(* Logix 5000 project; controller STAT 1756-L72 rev 20.12; software revision 20.04; part 16 of 34 *)
(* tags used below, declared in another part *)
   averflowput1 : DINT;
   averflowput2 : DINT;
   averK1 : DINT;
   averK2 : DINT;
   averL1 : DINT;
   averL2 : DINT;
   averL3 : DINT;
   averlpmpput2 : DINT;
   averpmpput1 : DINT;
   averQ1 : DINT;
   averQ2 : DINT;
   B16 : DINT[30];
   B17 : DINT[30];
   B3 : DINT[256];
   B9 : DINT[40];
   DateTime : DINT[7];   // DINT array tag for retrieve wallclock time through GSV created during conversion
   F8 : REAL[256];
   I19_000_Bit12 : ALIAS FOR I19[0].12;   // pulse puit put 1
   I19_000_Bit13 : ALIAS FOR I19[0].13;   // puit put 2
   I8_000_Bit09 : ALIAS FOR I8[0].9;   // midden niveau kuip 1 voorb. polyelectrolute
   I8_000_Bit10 : ALIAS FOR I8[0].10;   // hoog niveau kuip 1 voorb. polyelectrolute
   I8_000_Bit12 : ALIAS FOR I8[0].12;   // midden niveau kuip 2 voorb. polyelectrolute
   I8_000_Bit13 : ALIAS FOR I8[0].13;   // hoog niveau pekel
   N12 : DINT[230];
   N13 : DINT[230];
   N26 : DINT[256];
   O18_001_Bit02 : ALIAS FOR O18[1].2;   // pmp put 2
   O18_001_Bit04 : ALIAS FOR O18[1].4;   // PMP PUT 1
   pmpput1 : BOOL;
   pmpput2 : BOOL;
   T4 : TIMER[200];
   tot_put_1 : DINT;
   tot_put_2 : DINT;
(* ibt, continued *)

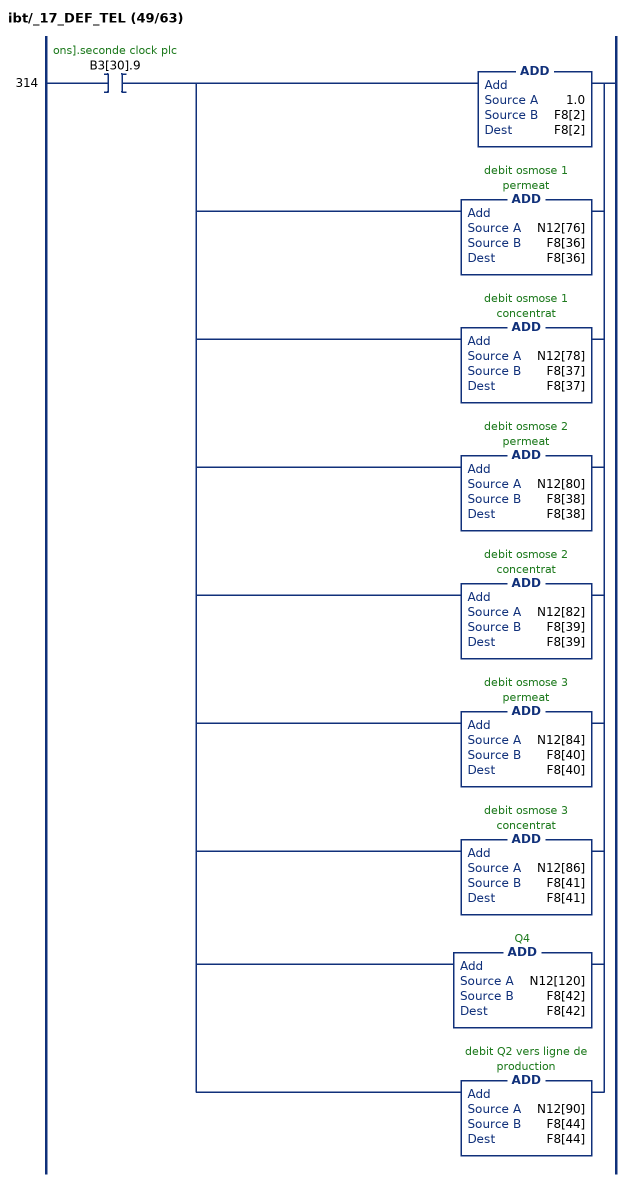
   [picture p273: ibt/_17_DEF_TEL rungs 314-314]
   314: XIC(B3[30].9)[ADD(1.0,F8[2],F8[2]) ,ADD(N12[76],F8[36],F8[36]) ,ADD(N12[78],F8[37],F8[37]) ,ADD(N12[80],F8[38],F8[38]) ,ADD(N12[82],F8[39],F8[39]) ,ADD(N12[84],F8[40],F8[40]) ,ADD(N12[86],F8[41],F8[41]) ,ADD(N12[120],F8[42],F8[42]) ,ADD(N12[90],F8[44],F8[44]) ];
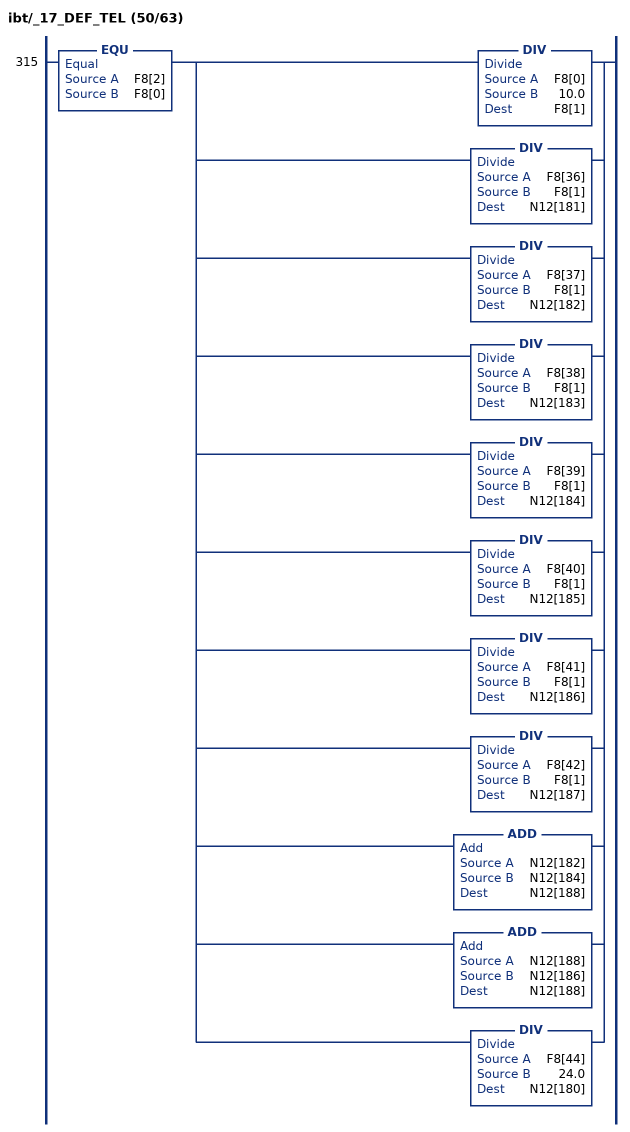
   315: EQU(F8[2],F8[0])[DIV(F8[0],10.0,F8[1]) ,DIV(F8[36],F8[1],N12[181]) ,DIV(F8[37],F8[1],N12[182]) ,DIV(F8[38],F8[1],N12[183]) ,DIV(F8[39],F8[1],N12[184]) ,DIV(F8[40],F8[1],N12[185]) ,DIV(F8[41],F8[1],N12[186]) ,DIV(F8[42],F8[1],N12[187]) ,ADD(N12[182],N12[184],N12[188]) ,ADD(N12[188],N12[186],N12[188]) ,DIV(F8[44],24.0,N12[180]) ];
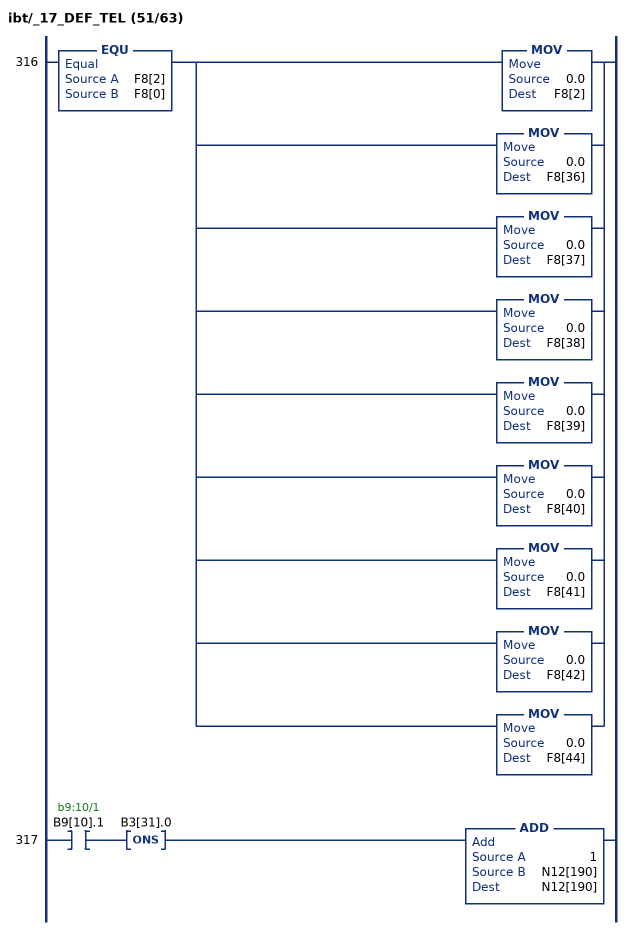
   316: EQU(F8[2],F8[0])[MOV(0.0,F8[2]) ,MOV(0.0,F8[36]) ,MOV(0.0,F8[37]) ,MOV(0.0,F8[38]) ,MOV(0.0,F8[39]) ,MOV(0.0,F8[40]) ,MOV(0.0,F8[41]) ,MOV(0.0,F8[42]) ,MOV(0.0,F8[44]) ];
   317: XIC(B9[10].1)ONS(B3[31].0)ADD(1,N12[190],N12[190]);
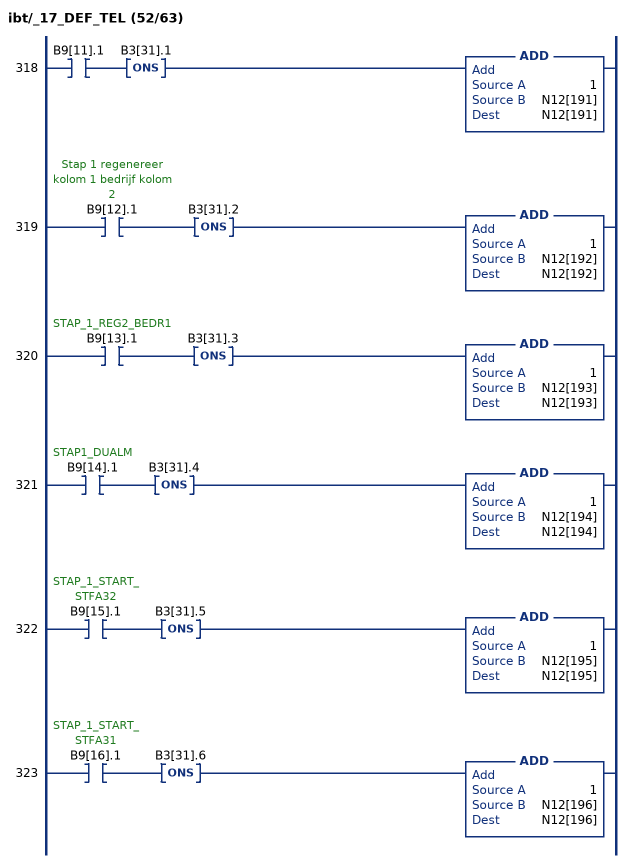
   318: XIC(B9[11].1)ONS(B3[31].1)ADD(1,N12[191],N12[191]);
   319: XIC(B9[12].1)ONS(B3[31].2)ADD(1,N12[192],N12[192]);
   320: XIC(B9[13].1)ONS(B3[31].3)ADD(1,N12[193],N12[193]);
   321: XIC(B9[14].1)ONS(B3[31].4)ADD(1,N12[194],N12[194]);
   322: XIC(B9[15].1)ONS(B3[31].5)ADD(1,N12[195],N12[195]);
   323: XIC(B9[16].1)ONS(B3[31].6)ADD(1,N12[196],N12[196]);
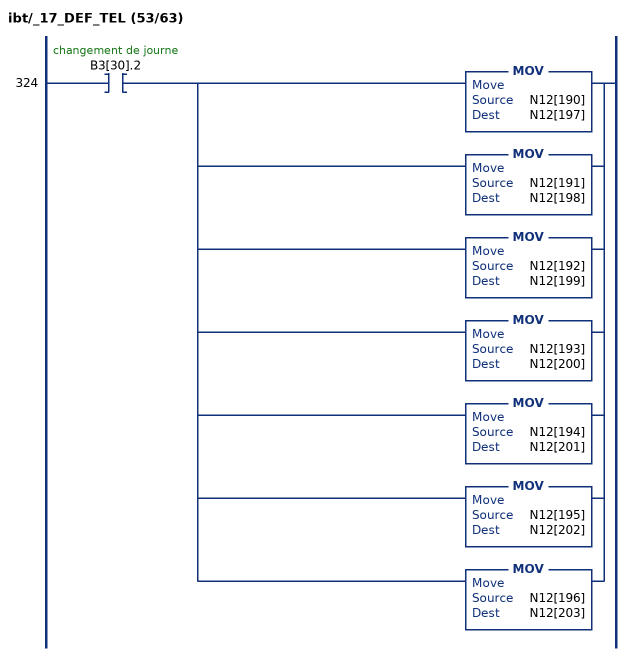
   324: XIC(B3[30].2)[MOV(N12[190],N12[197]) ,MOV(N12[191],N12[198]) ,MOV(N12[192],N12[199]) ,MOV(N12[193],N12[200]) ,MOV(N12[194],N12[201]) ,MOV(N12[195],N12[202]) ,MOV(N12[196],N12[203]) ];
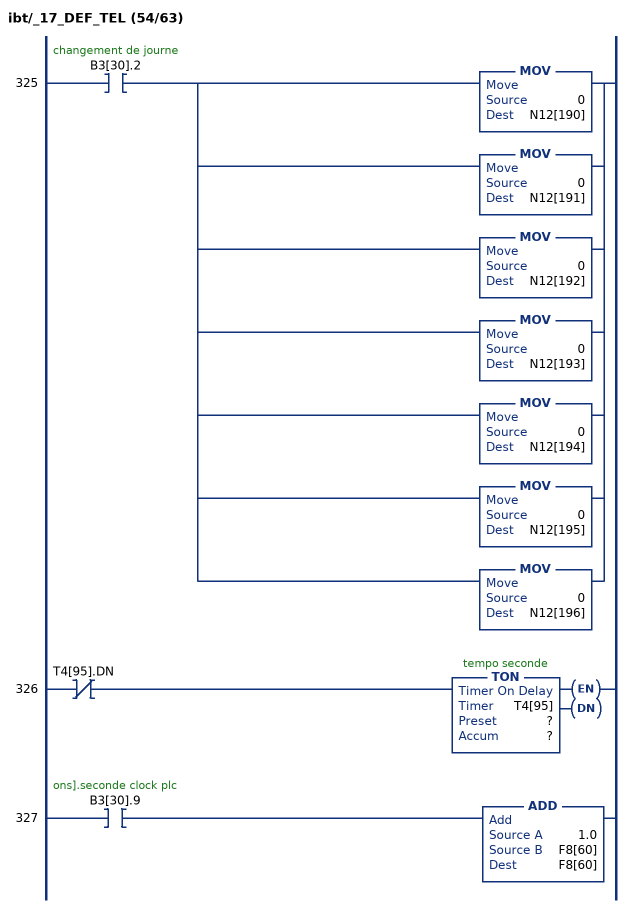
   325: XIC(B3[30].2)[MOV(0,N12[190]) ,MOV(0,N12[191]) ,MOV(0,N12[192]) ,MOV(0,N12[193]) ,MOV(0,N12[194]) ,MOV(0,N12[195]) ,MOV(0,N12[196]) ];
   326: XIO(T4[95].DN)TON(T4[95],?,?);
   327: XIC(B3[30].9)ADD(1.0,F8[60],F8[60]);
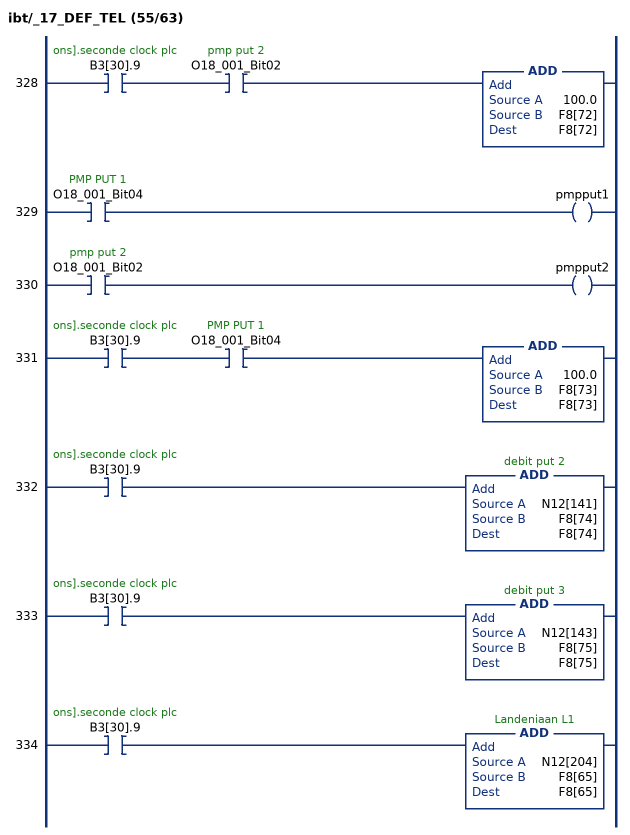
   328: XIC(B3[30].9)XIC(O18_001_Bit02)ADD(100.0,F8[72],F8[72]);
   329: XIC(O18_001_Bit04)OTE(pmpput1);
   330: XIC(O18_001_Bit02)OTE(pmpput2);
   331: XIC(B3[30].9)XIC(O18_001_Bit04)ADD(100.0,F8[73],F8[73]);
   332: XIC(B3[30].9)ADD(N12[141],F8[74],F8[74]);
   333: XIC(B3[30].9)ADD(N12[143],F8[75],F8[75]);
   334: XIC(B3[30].9)ADD(N12[204],F8[65],F8[65]);
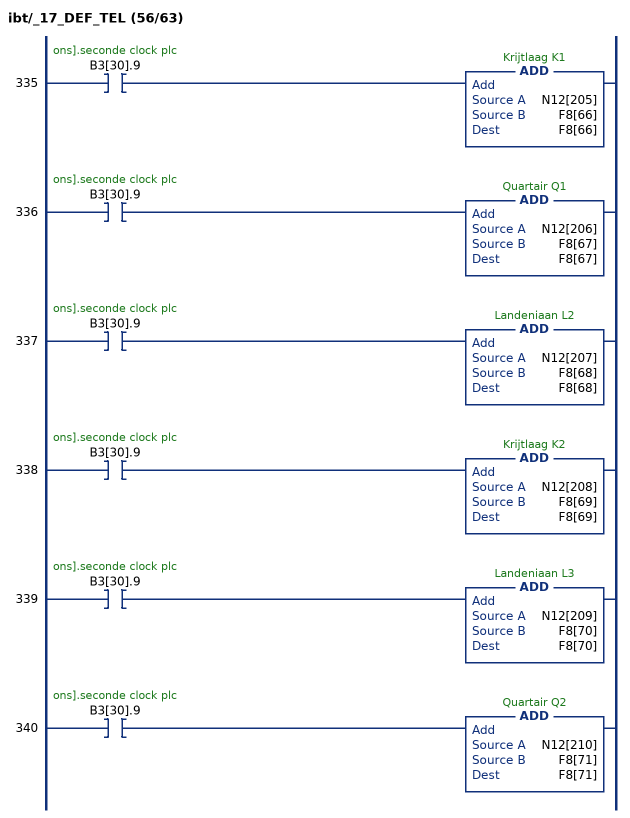
   335: XIC(B3[30].9)ADD(N12[205],F8[66],F8[66]);
   336: XIC(B3[30].9)ADD(N12[206],F8[67],F8[67]);
   337: XIC(B3[30].9)ADD(N12[207],F8[68],F8[68]);
   338: XIC(B3[30].9)ADD(N12[208],F8[69],F8[69]);
   339: XIC(B3[30].9)ADD(N12[209],F8[70],F8[70]);
   340: XIC(B3[30].9)ADD(N12[210],F8[71],F8[71]);
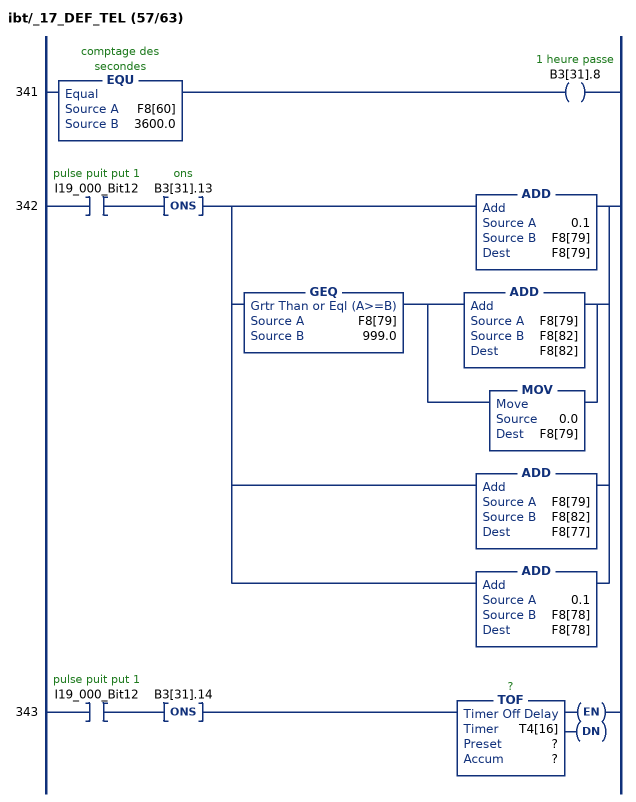
   341: EQU(F8[60],3600.0)OTE(B3[31].8);
   342: XIC(I19_000_Bit12)ONS(B3[31].13)[ADD(0.1,F8[79],F8[79]) ,GEQ(F8[79],999.0) [ADD(F8[79],F8[82],F8[82]) ,MOV(0.0,F8[79]) ] ,ADD(F8[79],F8[82],F8[77]) ,ADD(0.1,F8[78],F8[78]) ];
   343: XIC(I19_000_Bit12)ONS(B3[31].14)TOF(T4[16],?,?);
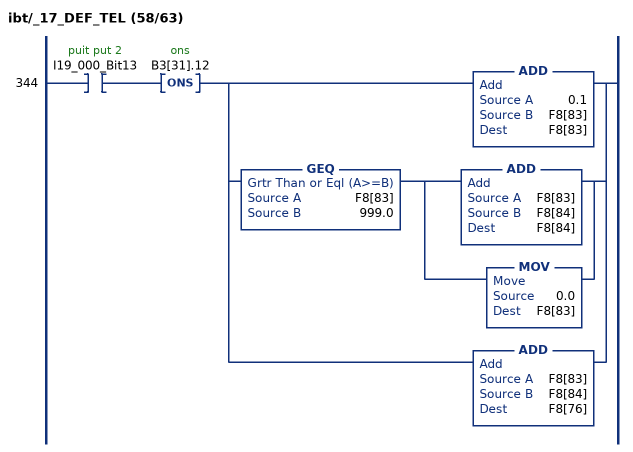
   344: XIC(I19_000_Bit13)ONS(B3[31].12)[ADD(0.1,F8[83],F8[83]) ,GEQ(F8[83],999.0) [ADD(F8[83],F8[84],F8[84]) ,MOV(0.0,F8[83]) ] ,ADD(F8[83],F8[84],F8[76]) ];
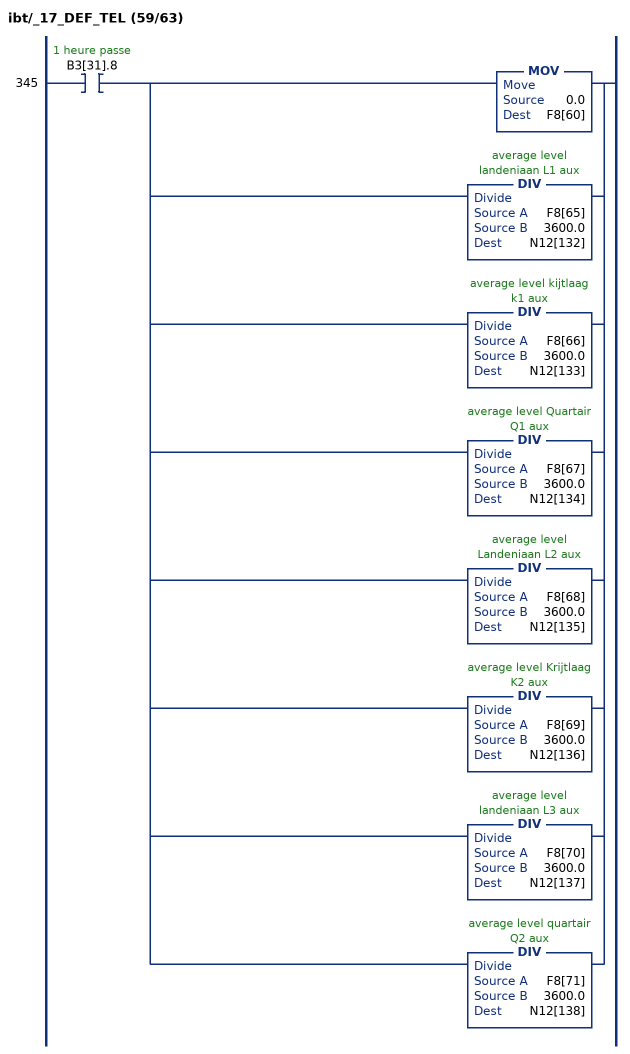
   345: XIC(B3[31].8)[MOV(0.0,F8[60]) ,DIV(F8[65],3600.0,N12[132]) ,DIV(F8[66],3600.0,N12[133]) ,DIV(F8[67],3600.0,N12[134]) ,DIV(F8[68],3600.0,N12[135]) ,DIV(F8[69],3600.0,N12[136]) ,DIV(F8[70],3600.0,N12[137]) ,DIV(F8[71],3600.0,N12[138]) ];
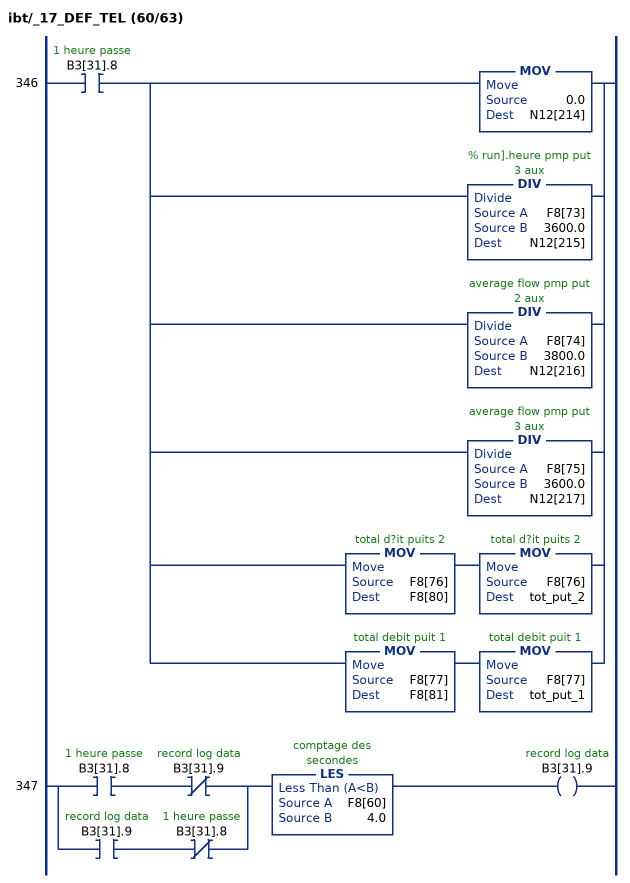
   346: XIC(B3[31].8)[MOV(0.0,N12[214]) ,DIV(F8[73],3600.0,N12[215]) ,DIV(F8[74],3800.0,N12[216]) ,DIV(F8[75],3600.0,N12[217]) ,MOV(F8[76],F8[80]) MOV(F8[76],tot_put_2) ,MOV(F8[77],F8[81]) MOV(F8[77],tot_put_1) ];
   347: [XIC(B3[31].8) XIO(B3[31].9) ,XIC(B3[31].9) XIO(B3[31].8) ]LES(F8[60],4.0)OTE(B3[31].9);
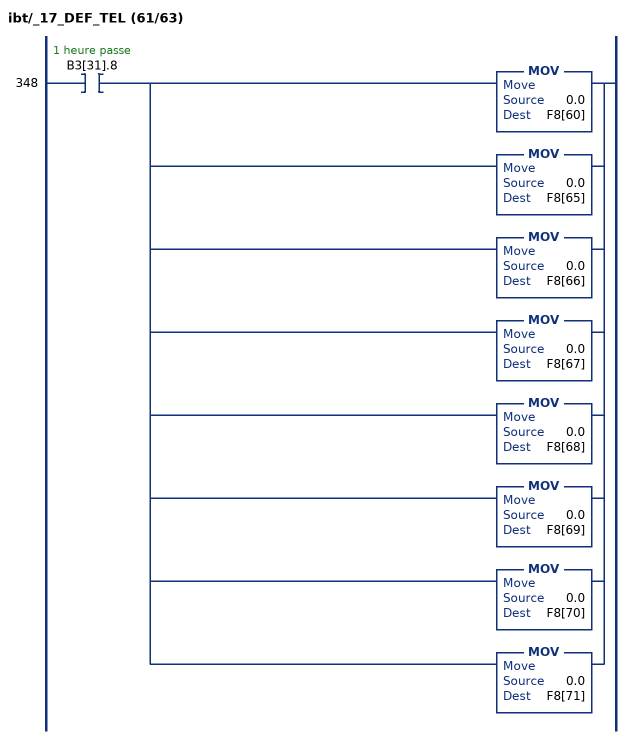
   348: XIC(B3[31].8)[MOV(0.0,F8[60]) ,MOV(0.0,F8[65]) ,MOV(0.0,F8[66]) ,MOV(0.0,F8[67]) ,MOV(0.0,F8[68]) ,MOV(0.0,F8[69]) ,MOV(0.0,F8[70]) ,MOV(0.0,F8[71]) ];
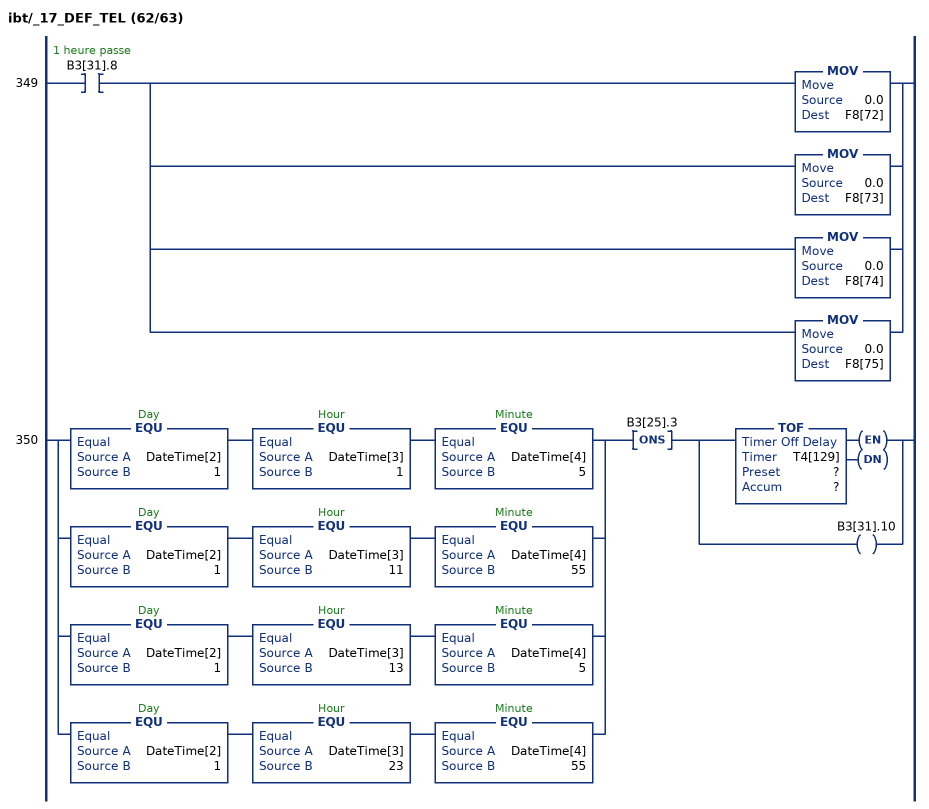
   349: XIC(B3[31].8)[MOV(0.0,F8[72]) ,MOV(0.0,F8[73]) ,MOV(0.0,F8[74]) ,MOV(0.0,F8[75]) ];
   350: [EQU(DateTime[2],1) EQU(DateTime[3],1) EQU(DateTime[4],5) ,EQU(DateTime[2],1) EQU(DateTime[3],11) EQU(DateTime[4],55) ,EQU(DateTime[2],1) EQU(DateTime[3],13) EQU(DateTime[4],5) ,EQU(DateTime[2],1) EQU(DateTime[3],23) EQU(DateTime[4],55) ]ONS(B3[25].3)[TOF(T4[129],?,?) ,OTE(B3[31].10) ];
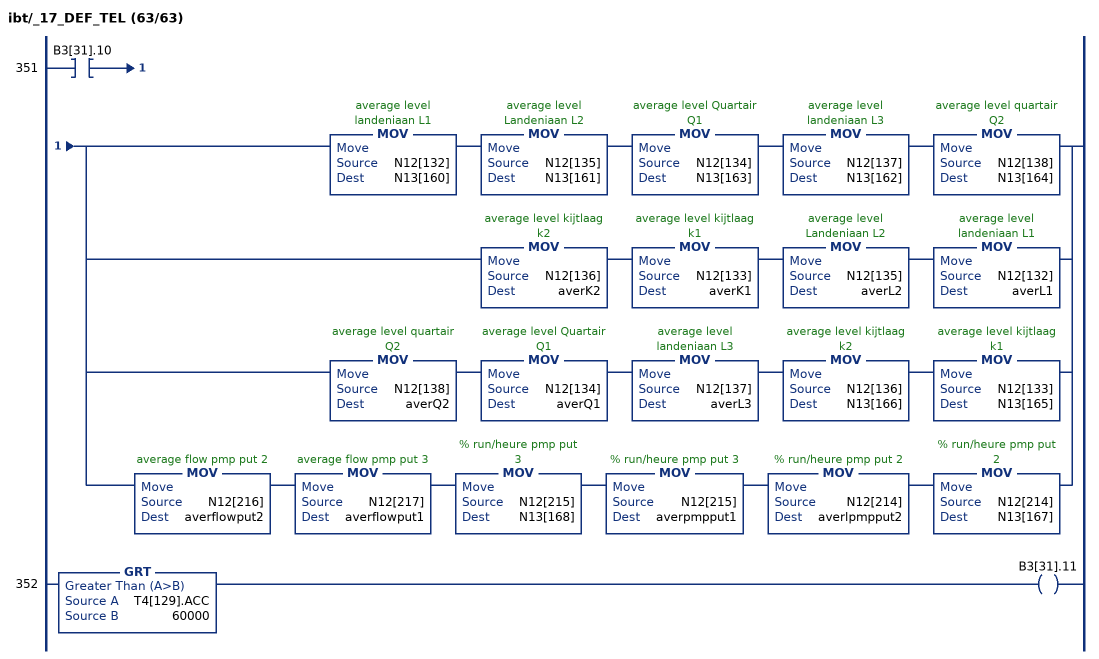
   351: XIC(B3[31].10)[MOV(N12[132],N13[160]) MOV(N12[135],N13[161]) MOV(N12[134],N13[163]) MOV(N12[137],N13[162]) MOV(N12[138],N13[164]) ,MOV(N12[136],averK2) MOV(N12[133],averK1) MOV(N12[135],averL2) MOV(N12[132],averL1) ,MOV(N12[138],averQ2) MOV(N12[134],averQ1) MOV(N12[137],averL3) MOV(N12[136],N13[166]) MOV(N12[133],N13[165]) ,MOV(N12[216],averflowput2) MOV(N12[217],averflowput1) MOV(N12[215],N13[168]) MOV(N12[215],averpmpput1) MOV(N12[214],averlpmpput2) MOV(N12[214],N13[167]) ];
   352: GRT(T4[129].ACC,60000)OTE(B3[31].11);
END_ROUTINE

ROUTINE _18_PAS_REI_Z   (* ladder *)
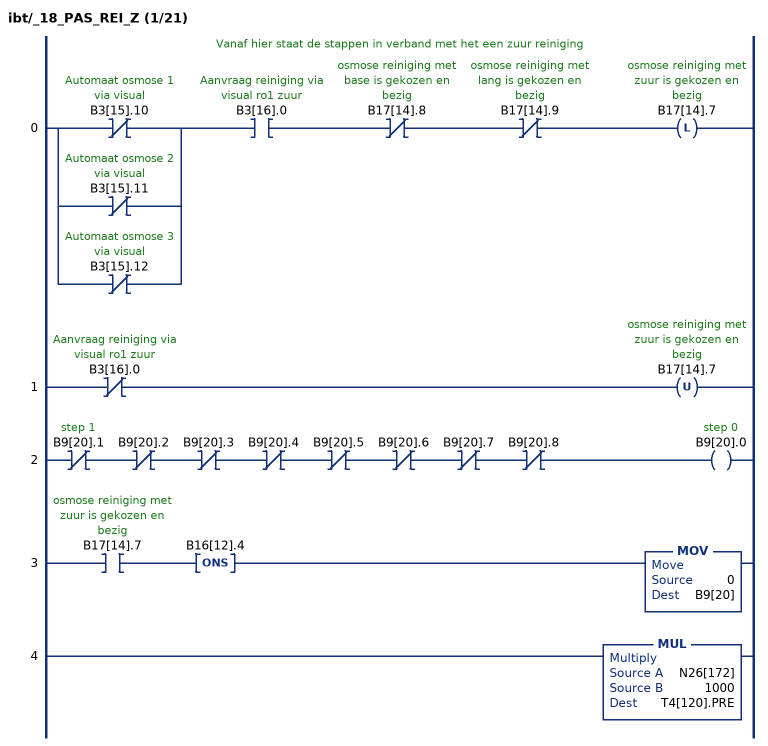
   // Vanaf hier staat de stappen in verband met het een zuur reiniging
   0: [XIO(B3[15].10) ,[XIO(B3[15].11) ,XIO(B3[15].12) ] ]XIC(B3[16].0)XIO(B17[14].8)XIO(B17[14].9)OTL(B17[14].7);
   1: XIO(B3[16].0)OTU(B17[14].7);
   2: XIO(B9[20].1)XIO(B9[20].2)XIO(B9[20].3)XIO(B9[20].4)XIO(B9[20].5)XIO(B9[20].6)XIO(B9[20].7)XIO(B9[20].8)OTE(B9[20].0);
   3: XIC(B17[14].7)ONS(B16[12].4)MOV(0,B9[20]);
   4: MUL(N26[172],1000,T4[120].PRE);
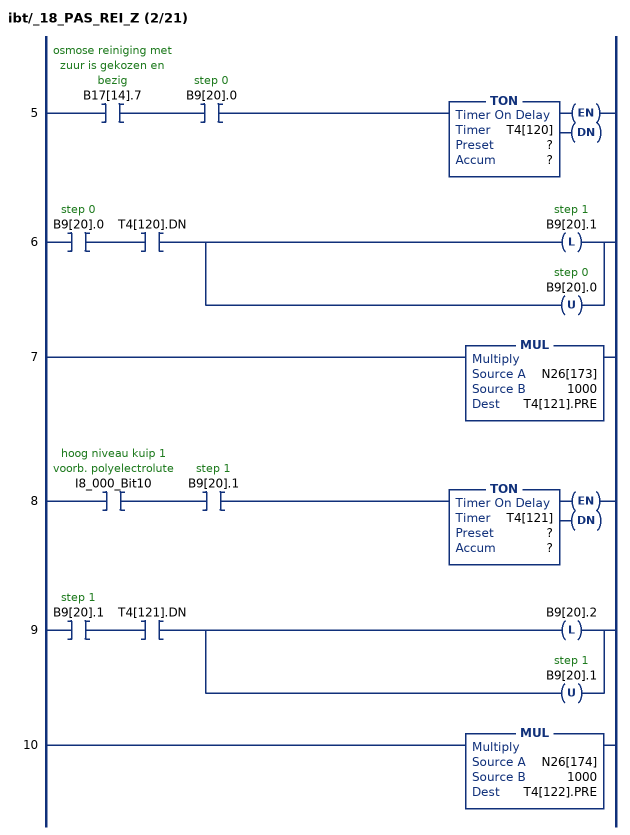
   5: XIC(B17[14].7)XIC(B9[20].0)TON(T4[120],?,?);
   6: XIC(B9[20].0)XIC(T4[120].DN)[OTL(B9[20].1) ,OTU(B9[20].0) ];
   7: MUL(N26[173],1000,T4[121].PRE);
   8: XIC(I8_000_Bit10)XIC(B9[20].1)TON(T4[121],?,?);
   9: XIC(B9[20].1)XIC(T4[121].DN)[OTL(B9[20].2) ,OTU(B9[20].1) ];
   10: MUL(N26[174],1000,T4[122].PRE);
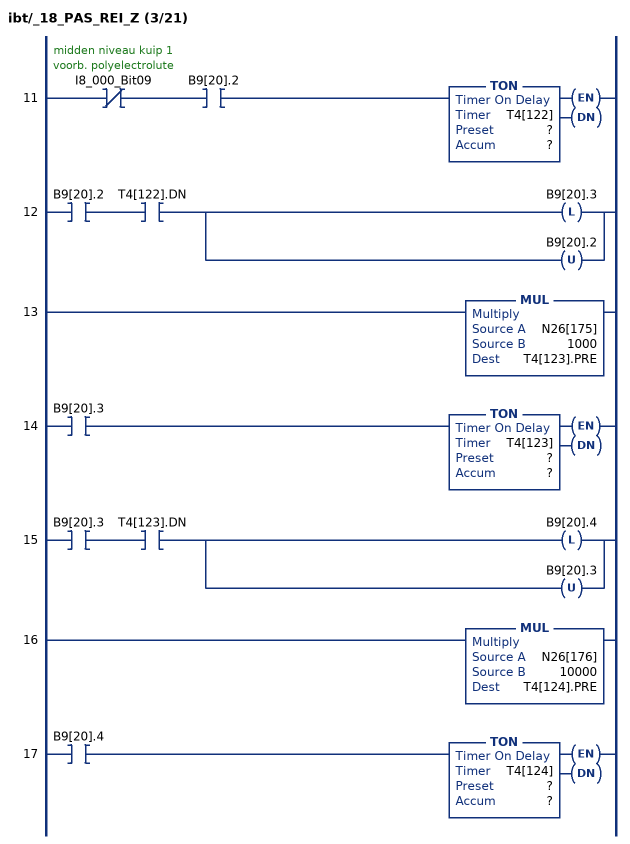
   11: XIO(I8_000_Bit09)XIC(B9[20].2)TON(T4[122],?,?);
   12: XIC(B9[20].2)XIC(T4[122].DN)[OTL(B9[20].3) ,OTU(B9[20].2) ];
   13: MUL(N26[175],1000,T4[123].PRE);
   14: XIC(B9[20].3)TON(T4[123],?,?);
   15: XIC(B9[20].3)XIC(T4[123].DN)[OTL(B9[20].4) ,OTU(B9[20].3) ];
   16: MUL(N26[176],10000,T4[124].PRE);
   17: XIC(B9[20].4)TON(T4[124],?,?);
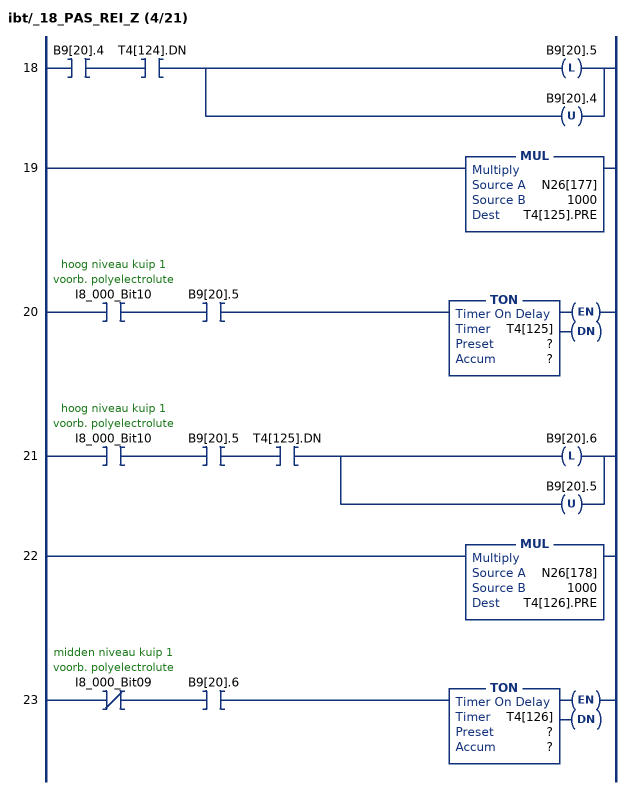
   18: XIC(B9[20].4)XIC(T4[124].DN)[OTL(B9[20].5) ,OTU(B9[20].4) ];
   19: MUL(N26[177],1000,T4[125].PRE);
   20: XIC(I8_000_Bit10)XIC(B9[20].5)TON(T4[125],?,?);
   21: XIC(I8_000_Bit10)XIC(B9[20].5)XIC(T4[125].DN)[OTL(B9[20].6) ,OTU(B9[20].5) ];
   22: MUL(N26[178],1000,T4[126].PRE);
   23: XIO(I8_000_Bit09)XIC(B9[20].6)TON(T4[126],?,?);
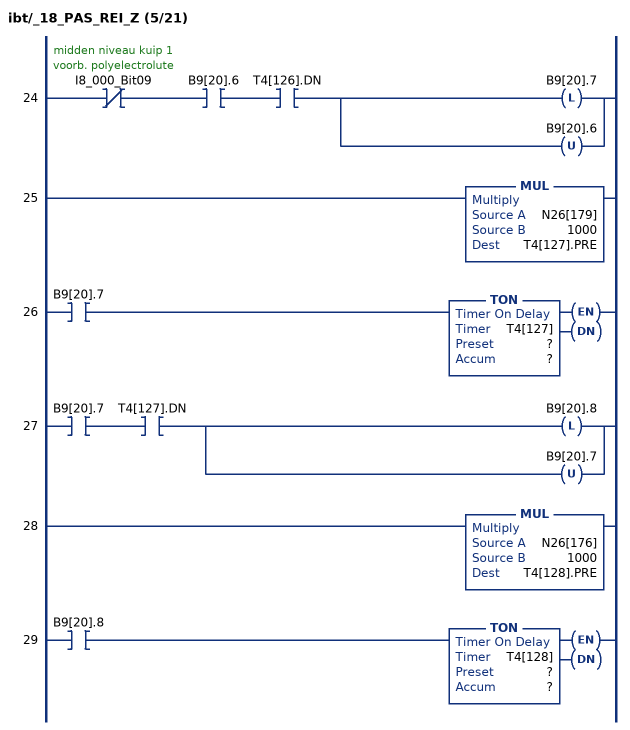
   24: XIO(I8_000_Bit09)XIC(B9[20].6)XIC(T4[126].DN)[OTL(B9[20].7) ,OTU(B9[20].6) ];
   25: MUL(N26[179],1000,T4[127].PRE);
   26: XIC(B9[20].7)TON(T4[127],?,?);
   27: XIC(B9[20].7)XIC(T4[127].DN)[OTL(B9[20].8) ,OTU(B9[20].7) ];
   28: MUL(N26[176],1000,T4[128].PRE);
   29: XIC(B9[20].8)TON(T4[128],?,?);
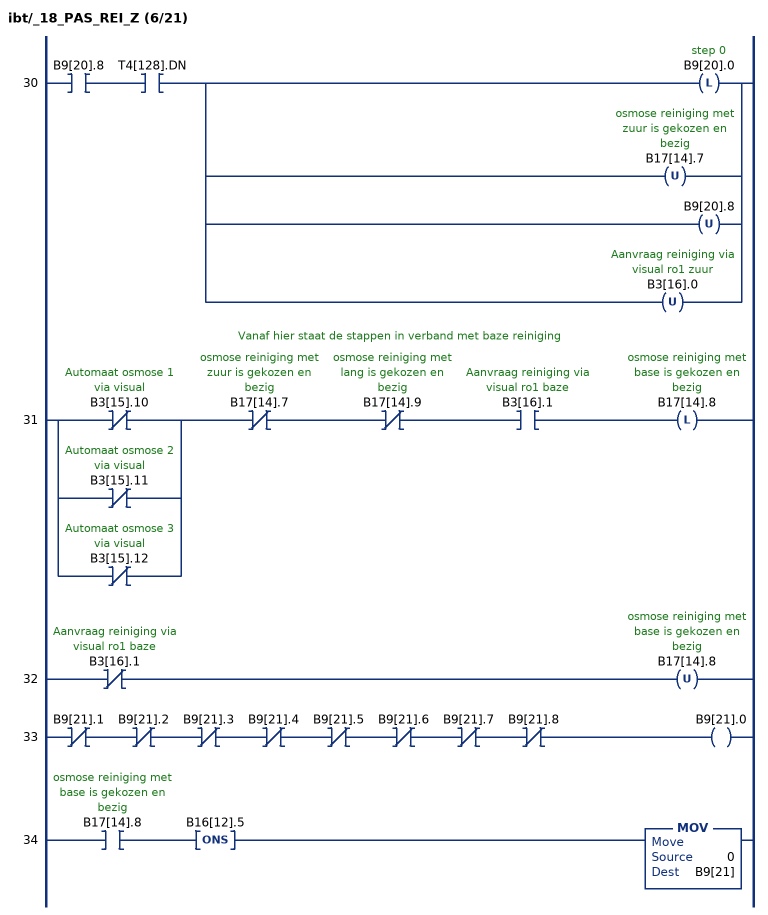
   30: XIC(B9[20].8)XIC(T4[128].DN)[[OTL(B9[20].0) ,OTU(B17[14].7) ] ,[OTU(B9[20].8) ,OTU(B3[16].0) ] ];
   // Vanaf hier staat de stappen in verband met baze reiniging
   31: [XIO(B3[15].10) ,[XIO(B3[15].11) ,XIO(B3[15].12) ] ]XIO(B17[14].7)XIO(B17[14].9)XIC(B3[16].1)OTL(B17[14].8);
   32: XIO(B3[16].1)OTU(B17[14].8);
   33: XIO(B9[21].1)XIO(B9[21].2)XIO(B9[21].3)XIO(B9[21].4)XIO(B9[21].5)XIO(B9[21].6)XIO(B9[21].7)XIO(B9[21].8)OTE(B9[21].0);
   34: XIC(B17[14].8)ONS(B16[12].5)MOV(0,B9[21]);
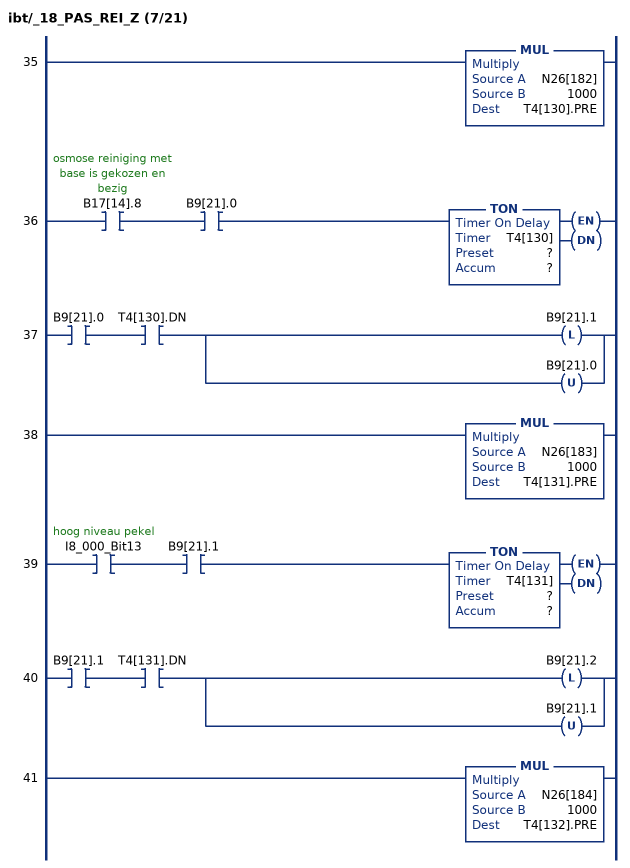
   35: MUL(N26[182],1000,T4[130].PRE);
   36: XIC(B17[14].8)XIC(B9[21].0)TON(T4[130],?,?);
   37: XIC(B9[21].0)XIC(T4[130].DN)[OTL(B9[21].1) ,OTU(B9[21].0) ];
   38: MUL(N26[183],1000,T4[131].PRE);
   39: XIC(I8_000_Bit13)XIC(B9[21].1)TON(T4[131],?,?);
   40: XIC(B9[21].1)XIC(T4[131].DN)[OTL(B9[21].2) ,OTU(B9[21].1) ];
   41: MUL(N26[184],1000,T4[132].PRE);
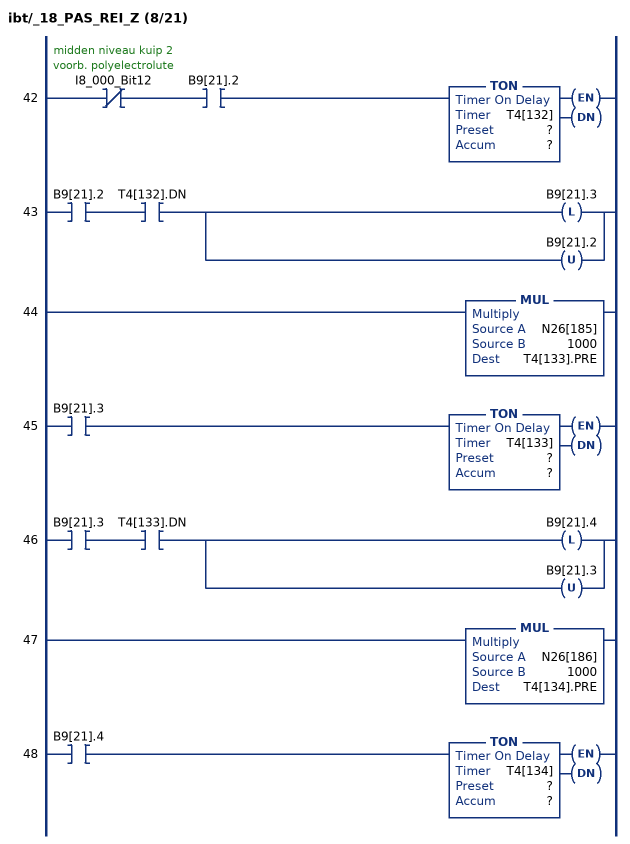
   42: XIO(I8_000_Bit12)XIC(B9[21].2)TON(T4[132],?,?);
   43: XIC(B9[21].2)XIC(T4[132].DN)[OTL(B9[21].3) ,OTU(B9[21].2) ];
   44: MUL(N26[185],1000,T4[133].PRE);
   45: XIC(B9[21].3)TON(T4[133],?,?);
   46: XIC(B9[21].3)XIC(T4[133].DN)[OTL(B9[21].4) ,OTU(B9[21].3) ];
   47: MUL(N26[186],1000,T4[134].PRE);
   48: XIC(B9[21].4)TON(T4[134],?,?);
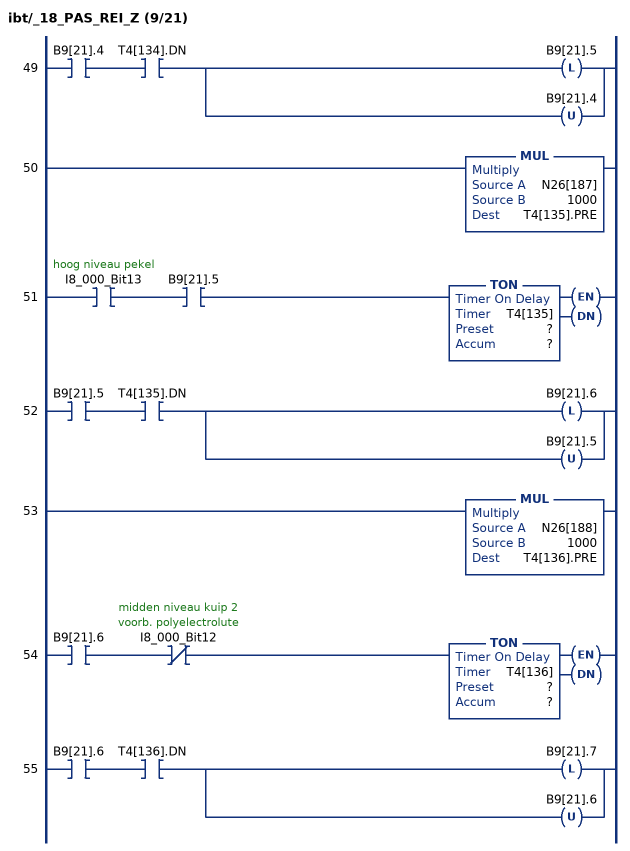
   49: XIC(B9[21].4)XIC(T4[134].DN)[OTL(B9[21].5) ,OTU(B9[21].4) ];
   50: MUL(N26[187],1000,T4[135].PRE);
   51: XIC(I8_000_Bit13)XIC(B9[21].5)TON(T4[135],?,?);
   52: XIC(B9[21].5)XIC(T4[135].DN)[OTL(B9[21].6) ,OTU(B9[21].5) ];
   53: MUL(N26[188],1000,T4[136].PRE);
   54: XIC(B9[21].6)XIO(I8_000_Bit12)TON(T4[136],?,?);
   55: XIC(B9[21].6)XIC(T4[136].DN)[OTL(B9[21].7) ,OTU(B9[21].6) ];
